SUBAPPLICATION Ventilsteuerung_Uebung_016 (* Background Colour umschalten *)
  (* Standard: 61499-2 *)
  (* Version 1.0, 2023-10-23, franz *)
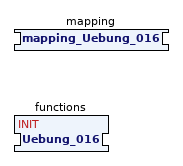
  SUBAPPS
    mapping : mapping_Uebung_016;
    functions : Uebung_016;
  END_SUBAPPS
END_SUBAPPLICATION
